# EPICS substitutions: apps/caenHvApp/Db/mvtOnOff-fmt.substitutions
file "db/mvtOnOff-fmt-1type.db"
{
    pattern { INOUT TYPE  PW    PWVAL}
            { ""    DRIFT pwoff 0 }
            { ""    DRIFT pwon  1 }
            { IN_   STRIP pwoff 0 }
            { IN_   STRIP pwon  1 }
            { OUT_  STRIP pwoff 0 }
            { OUT_  STRIP pwon  1 }
}
